TYPE ST_NameValue :
STRUCT
	sName 	: STRING(31);
	sValue 	: STRING; 
END_STRUCT
END_TYPE

(* stored: Version 1.1.0.1
   DUT ST_NameValue: Id {666ee2f4-fb66-411f-8da6-a6ddabea0c86} *)
